FUNCTION_BLOCK aiSignalDecode (* Basic Function Block Type *)
  (* Standard: 61499-2 *)
  (* Version 0.0, 7/8/2026, Schneider Electric, Template *)
  PACKAGE SE.Nereda;
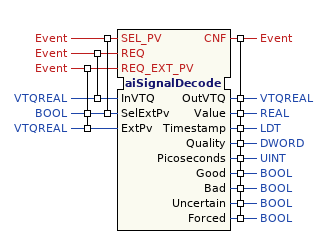
  EVENT_INPUT
    SEL_PV WITH SelExtPv;
    REQ WITH InVTQ; (* Normal Execution Request *)
    REQ_EXT_PV WITH SelExtPv, ExtPv;
  END_EVENT
  EVENT_OUTPUT
    CNF WITH OutVTQ, Value, Timestamp, Quality, Picoseconds, Good, Bad, Uncertain, Forced; (* Execution Confirmation *)
  END_EVENT
  VAR_INPUT
    InVTQ : VTQREAL;
    SelExtPv : BOOL;
    ExtPv : VTQREAL;
  END_VAR
  VAR_OUTPUT
    OutVTQ : VTQREAL;
    Value : REAL;
    Timestamp : LDT;
    Quality : DWORD;
    Picoseconds : UINT;
    Good : BOOL;
    Bad : BOOL;
    Uncertain : BOOL;
    Forced : BOOL;
  END_VAR
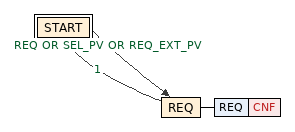
  EC_STATES
    START; (* Initial State *)
    REQ : REQ -> CNF; (* Normal execution *)
  END_STATES
  EC_TRANSITIONS
    START TO REQ := REQ OR SEL_PV OR REQ_EXT_PV;
    REQ TO START := 1;
  END_TRANSITIONS
  ALGORITHM REQ IN ST: (* Normally executed algorithm *)
;
IF SelExtPv THEN
    OutVTQ:= ExtPv;
ELSE
    OutVTQ:= InVTQ;
END_IF;


Value := InVTQ.value;
Picoseconds := InVTQ.picosecs;
Quality := InVTQ.quality;
Timestamp := InVTQ.timestamp;

IF Quality = 16#960000 THEN
    Good:=FALSE;
    Uncertain := FALSE;
	Bad := FALSE;
    Forced := TRUE;
ELSIF Quality >= 16#00000000 AND Quality <= 16#3FFFFFFF THEN
    Good:=TRUE;
    Uncertain := FALSE;
	Bad := FALSE;
    Forced := FALSE;
ELSIF Quality >= 16#40000000 AND Quality <= 16#7FFFFFFF THEN
    Good:=FALSE;
    Uncertain := TRUE;
	Bad := FALSE;
    Forced := FALSE;
ELSIF Quality >= 16#80000008 THEN
    Good:=FALSE;
    Uncertain := FALSE;
	Bad := TRUE;
    Forced := FALSE;
END_IF;
  END_ALGORITHM
END_FUNCTION_BLOCK
